Staubli VAL3: readNumValue.pgx

public program readNumValue(num x_nHandle, string x_sCol, num x_nRow, num& value_[], bool& x_bResult[])
  local bool l_bIsOK
  local string strValue
  local string strDummy
  local string l_sCellNumber
begin
  // modified  7.03.2008
  //------------------------------------------------------------
  // Check format of the cell to read
  l_sCellNumber=x_sCol+toString("",x_nRow)
  call CheckCellFormat(l_sCellNumber,l_bIsOK)
  if l_bIsOK
    // read contents of cell and transform it to a numerical value
    //? "CellValue : "+l_sCellNumber
    call readStrValue(x_nHandle,l_sCellNumber,strValue,x_bResult)
    if x_bResult
      strDummy=toNum(strValue,value_,x_bResult)
      if !x_bResult
        errorCode[x_nHandle]=3
      endIf
    endIf
  else
    errorCode[x_nHandle]=4
    x_bResult=false
  endIf
end
